(*********************************** G.D S.p.A. - Technical Department ***********************************
============= PROGRAM INFO ============
FOLDER:             TBD
MACHINES INVOLVED:  TBD 

============= DESCRIPTION =============
CSP machine declaration

============= REVISIONS ===============
Date		Version	 	Author      	Description             
----------	-------		------------  	--------------------------------------------
2019/04/05 	0000.00	 	M.Grasso		Creation of the PRG

**********************************************************************************************************)
(*$R process_ref := prc; $*)
PROGRAM csp_case_feed_reject_accU
VAR
		
	prc:											process;
	prc_path:										STRING;
	
END_VAR

_read_var_input();

_object_manager();

IF NOT objects_running()
THEN
	RETURN;	
END_IF

_read_process_image();

_mode_manager();

_set_runtime_properties();

(********************************* BODY *********************************)
(* MACHINE COMMANDS *)
(************************************************************************)

_handle_messages();

_write_output();

ACTION _handle_messages:
;
END_ACTION

ACTION _handle_process_test:
;
END_ACTION

ACTION _mode_manager:
IF process_mode_req_is_pending(prc)
THEN
    process_apply_mode_req_first_step(prc);
    CASE process_get_mode(prc) OF
        MODE_TO_ABSENT:
			;
        MODE_TO_INACTIVE:
			;
        MODE_TO_TEST:
			;
        MODE_TO_OPERATIONAL:
			;
    END_CASE
    process_apply_mode_req_second_step(prc);
END_IF
END_ACTION

ACTION _object_manager:
IF objects_initialization()
THEN
	sub_process_init(
		object_name					:= 'csp_case_feed_reject_accU.prc', 
		process						:= csp_case_feed_reject.prc, 
		CONVERSION_this				:= prc);
		
	prc_path 						:= process_get_path(prc);
END_IF

IF objects_running()
THEN
	process_cycle(prc);
END_IF
END_ACTION

ACTION _read_process_image:
;
END_ACTION

ACTION _read_var_input:
;
END_ACTION

ACTION _set_runtime_properties:
;
END_ACTION

ACTION _write_output:
;
END_ACTION

END_PROGRAM

(* stored: Version 1.1.0.1, ProductVersion 3.1.4024.3
   POU csp_case_feed_reject_accU: Id {729391a4-1535-4823-bbab-02f2b3785663}, SpecialFunc None
   Action _handle_messages: Id {5974abf1-f5c8-4af4-a434-84cce4ba5e31}
   Action _handle_process_test: Id {67e1eb0a-4969-416f-b533-0a2438db36c7}
   Action _mode_manager: Id {183d61ed-95b0-4e85-a763-f9ff053adb77}
   Action _object_manager: Id {ed657445-78a0-4c1a-9c81-e456d2bba472}
   Action _read_process_image: Id {0e09e3b0-3513-4c1f-9c75-da8040c3cbc5}
   Action _read_var_input: Id {721e5ee0-5553-49d4-a804-d4fd61dc3a1d}
   Action _set_runtime_properties: Id {0eed959d-1fb0-4d2e-affa-4634bf782caf}
   Action _write_output: Id {b0cb365e-8678-4905-b4f7-d010bffac732} *)
